FUNCTION_BLOCK FB_Filter_LowPass
VAR_INPUT
END_VAR
VAR_OUTPUT
END_VAR
VAR
END_VAR

END_FUNCTION_BLOCK

(* stored: Version 1.1.0.1, ProductVersion 3.1.4024.13
   POU FB_Filter_LowPass: Id {09a317c6-1b69-42ae-bf7c-6979c46a34ca}, SpecialFunc None *)
